// TIA Portal V18 export
// export: Created 2026-03-12T15:56:20.3071376Z, ExportSetting WithDefaults, DisplayName Totally Integrated Automation Portal, DisplayVersion V18 Update 5, DisplayName TIA Portal Openness, DisplayVersion V18 Update 5, DisplayName TIA Portal Version Control Interface, DisplayVersion V18, DisplayName SINAMICS Startdrive Advanced, DisplayVersion V18, DisplayName SINAMICS Startdrive G130, G150, S120, S150, SINAMICS MV, S210, DisplayVersion V18, DisplayName SINAMICS Startdrive G110M, G120, G120C, G120D, G120P, G115D, DisplayVersion V18, DisplayName STEP 7 Professional, DisplayVersion V18 Update 5, DisplayName STEP 7 Safety, DisplayVersion V18, DisplayName WinCC Professional, DisplayVersion V18 Update 5
DATA_BLOCK "FB CONDIÇÃO DE PARTIDA BH-01B"   // DB217
VERSION : 0.1
// stored: AutoNumber true, DBAccessibleFromOPCUA true, DBAccessibleFromWebserver true, InstanceOfName FB CONDIÇÃO DE PARTIDA, InstanceOfType FB
"FB CONDIÇÃO DE PARTIDA"
   // VAR_INPUT
   //    INPUT_LIGADO : Bool;
   //    INPUT_DESLIGADO : Bool;
   //    INPUT_FALHA : Bool;
   //    INPUT_LOCAL : Bool;
   //    INPUT_REMOTO : Bool;
   //    INPUT_LOC_AUTO : Bool;
   //    INPUT_FALHA_PROFINET : Bool;
   //    INPUT_HABILITA_LIGA_AUTO : Bool;
   //    CMD_LIGA : Bool;
   //    CMD_MANUTEN : Bool;
   //    CMD_MODO : Bool;
   // END_VAR
   // VAR_OUTPUT
   //    STATUS_MOTOR : Byte;
   //    LIGA_BOMBA : Bool;
   //    REMOTO_MAN : Bool;
   //    REMOTO_AUTO : Bool;
   //    LOCAL_MAN : Bool;
   // END_VAR
   // VAR
   //    MANUTEN : Bool;
   //    REMOTO : Bool;
   //    FALHA : Bool;
   //    LOCAL_AUTO : Bool;
   //    LIGA_REM_MAN : Bool;
   //    LIGA_REM_AUTO : Bool;
   // END_VAR
BEGIN
END_DATA_BLOCK
